FUNCTION TIMEMUL : TIME
VAR_INPUT
	TIME_IN: TIME;
	VALUE: REAL;
END_VAR
VAR
END_VAR
VAR // added by the converter: edge detectors and wires of the graphical bodies
    _w1 : REAL;
END_VAR

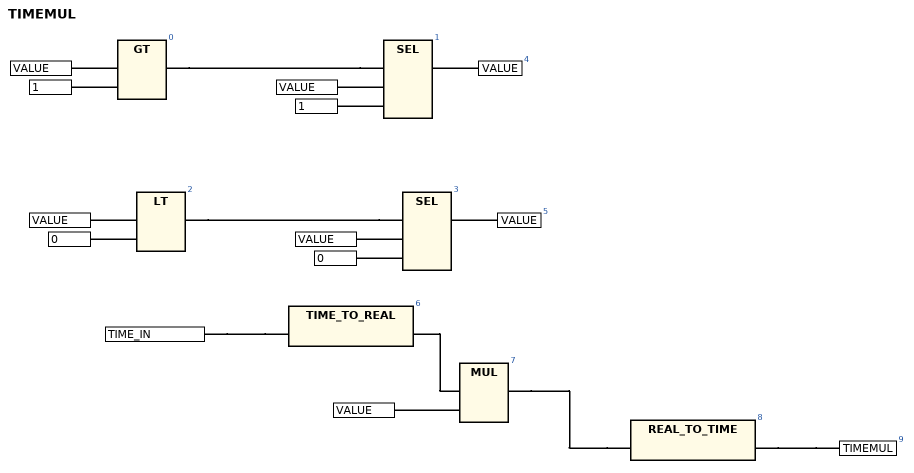
_w1 := SEL(VALUE < 0, VALUE, 0);
VALUE := SEL(VALUE > 1, VALUE, 1);
VALUE := _w1;
TIMEMUL := REAL_TO_TIME(TIME_TO_REAL(TIME_IN) * VALUE);

END_FUNCTION

(* stored: Version 1.1.0.1, ProductVersion 3.1.4024.12
   POU TIMEMUL: Id {55a7f7f6-0eb7-4ff5-80b1-efe179e97be3}, SpecialFunc None *)
